TYPE
  (* Standard: 61499-1 *)
  (* Version 1.0, 2026-07-21, Dimitrios Kalligaridis *)
  PACKAGE mypackage;
  RepairStruct : STRUCT
    keep : BOOL;
    other : BOOL;
  END_STRUCT;
END_TYPE
